(* PLC project Unnamed, 不明 Unnamed 1 *)
(* stored: creationDateTime 2022-12-26T15:45:20, modificationDateTime 2022-12-30T15:52:11 *)

PROGRAM prog
  VAR
    LED AT %QX0.0 : BOOL;  (* 7番ポート *)
  END_VAR
  VAR
    Timer : TIME := T#500ms;  (* 0.5秒 *)
    TimeOn : TON;
    TimeOff : TOF;
  END_VAR

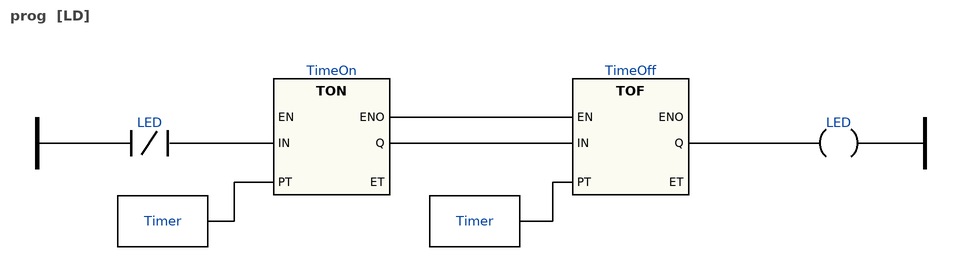
(* LD diagram, written out as Structured Text *)
TimeOn(IN := NOT LED, PT := Timer);
TimeOff(EN := TimeOn.ENO, IN := TimeOn.Q, PT := Timer);
LED := TimeOff.Q;
END_PROGRAM

CONFIGURATION Config0
  RESOURCE Res0 ON PLC
    TASK task0(INTERVAL := T#20ms, PRIORITY := 0);
    PROGRAM instance0 WITH task0 : prog;
  END_RESOURCE
END_CONFIGURATION
